% RSLogix 500 project I2P Job 11 Alexander_Loynd.RSS, saved by version 10.00.00.00 %
PROJECT "ML06A"    % processor: Bul.1763 MicroLogix 1100 Series B %

PROGRAM FILES
  LAD 2   7 rungs

DATA FILES
  O0 OUTPUT  4 elements
  I1 INPUT  6 elements
  S2 STATUS  66 elements
  B3 BINARY  1 elements
  T4 TIMER  1 elements
  C5 COUNTER  1 elements
  R6 CONTROL  1 elements
  N7 INTEGER  1 elements
  F8 FLOAT  1 elements

LADDER 2
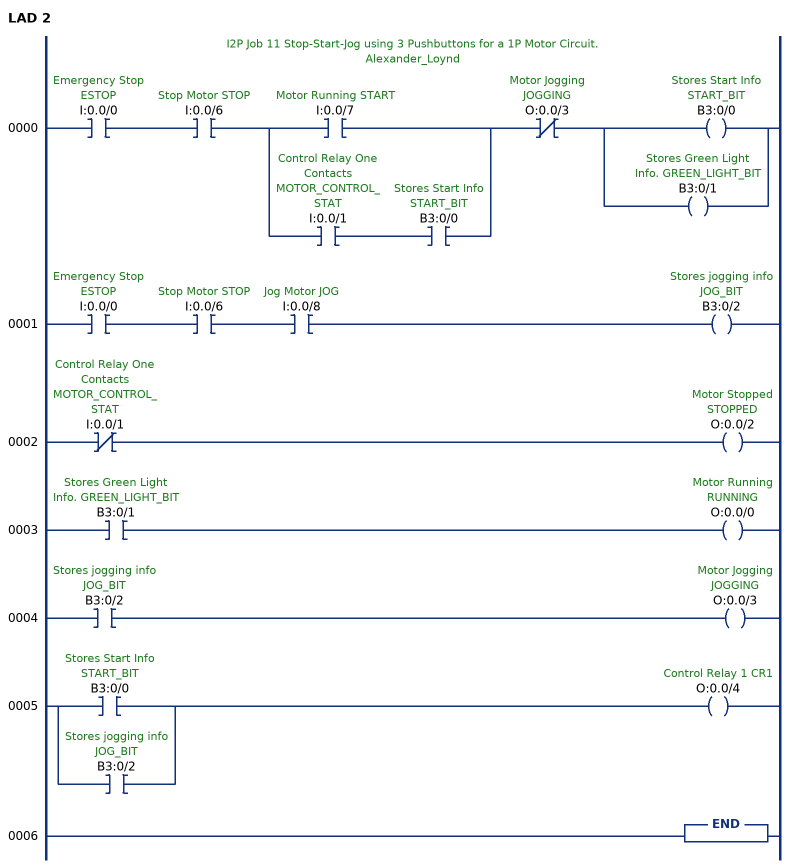
% Rung: 0 %
% I2P Job 11 Stop-Start-Jog using 3 Pushbuttons for a 1P Motor Circuit.
% Alexander_Loynd %
SOR XIC I:0.0/0 XIC I:0.0/6 BST XIC I:0.0/7 NXB XIC I:0.0/1 XIC B3:0/0 BND XIO O:0.0/3 BST OTE B3:0/0 NXB OTE B3:0/1 BND EOR
%   I:0.0/0  ESTOP  "Emergency Stop" %
%   I:0.0/6  STOP  "Stop Motor" %
%   I:0.0/7  START  "Motor Running" %
%   I:0.0/1  MOTOR_CONTROL_STAT  "Control Relay One Contacts" %
%   B3:0/0  START_BIT  "Stores Start Info" %
%   O:0.0/3  JOGGING  "Motor Jogging" %
%   B3:0/1  GREEN_LIGHT_BIT  "Stores Green Light Info." %
% Rung: 1 %
SOR XIC I:0.0/0 XIC I:0.0/6 XIC I:0.0/8 OTE B3:0/2 EOR
%   I:0.0/0  ESTOP  "Emergency Stop" %
%   I:0.0/6  STOP  "Stop Motor" %
%   I:0.0/8  JOG  "Jog Motor" %
%   B3:0/2  JOG_BIT  "Stores jogging info" %
% Rung: 2 %
SOR XIO I:0.0/1 OTE O:0.0/2 EOR
%   I:0.0/1  MOTOR_CONTROL_STAT  "Control Relay One Contacts" %
%   O:0.0/2  STOPPED  "Motor Stopped" %
% Rung: 3 %
SOR XIC B3:0/1 OTE O:0.0/0 EOR
%   B3:0/1  GREEN_LIGHT_BIT  "Stores Green Light Info." %
%   O:0.0/0  RUNNING  "Motor Running" %
% Rung: 4 %
SOR XIC B3:0/2 OTE O:0.0/3 EOR
%   B3:0/2  JOG_BIT  "Stores jogging info" %
%   O:0.0/3  JOGGING  "Motor Jogging" %
% Rung: 5 %
SOR BST XIC B3:0/0 NXB XIC B3:0/2 BND OTE O:0.0/4 EOR
%   B3:0/0  START_BIT  "Stores Start Info" %
%   B3:0/2  JOG_BIT  "Stores jogging info" %
%   O:0.0/4  CR1  "Control Relay 1" %
% Rung: 6 %
SOR END EOR

OTHER DOCUMENTED ADDRESSES
  I:0.0/2  CR2_STAT  "Control Relay Two Contacts"
  I:0.0/3  3PSS_A  "Three Position Selector Switch A Position"
  I:0.0/4  3PSS_B  "Three Position Selector Switch B Posistion"
  I:0.0/5  2PSS  "Two Position Selector Switch"
  O:0.0/1  YPL  "Yellow Pilot Light"
  O:0.0/5  CR2  "Control Relay 2"
